Staubli VAL3: create_sphere.pgx

public program create_sphere(point x_pOrigin, num x_nRadius)
begin
  //
  // build the sphere
  //
  // Origin
  pOrigin_sphere.trsf=position(x_pOrigin,world)
  bCreate_sphere=true
  // Radius
  nRadius_sphere=x_nRadius
end
